FUNCTION_BLOCK CylinderSA (* Composite Function Block Type *)
  (* Standard: 61499-2 *)
  (* Version 0.0, 5/26/2016, Andrei, nxtControl GmbH, template *)
  PACKAGE Main;
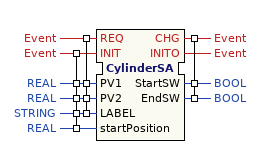
  EVENT_INPUT
    REQ WITH PV1, PV2, LABEL; (* Normal Execution Request *)
    INIT WITH PV1, PV2, LABEL, startPosition; (* Initialization Request *)
  END_EVENT
  EVENT_OUTPUT
    CHG WITH StartSW, EndSW;
    INITO; (* Initialization Confirm *)
  END_EVENT
  VAR_INPUT
    PV1 : REAL; (* Input event qualifier *)
    PV2 : REAL;
    LABEL : STRING;
    startPosition : REAL;
  END_VAR
  VAR_OUTPUT
    StartSW : BOOL; (* Output event qualifier *)
    EndSW : BOOL;
  END_VAR
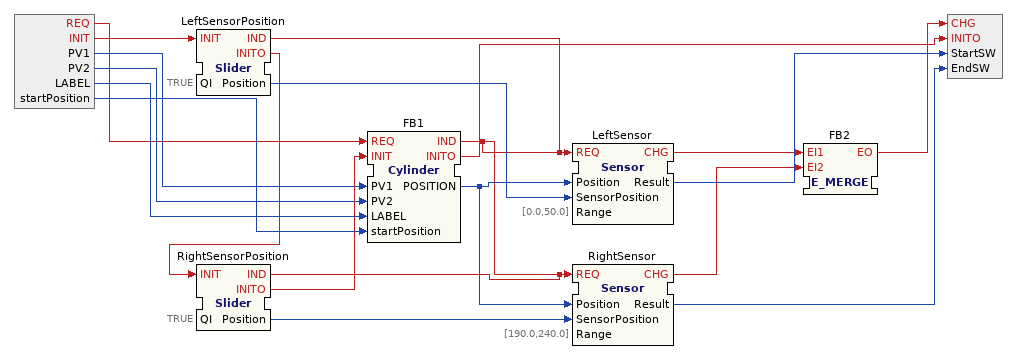
  FBS
    FB2 : E_MERGE;
    FB1 : Cylinder;
    LeftSensorPosition : Slider(QI := TRUE);
    RightSensorPosition : Slider(QI := TRUE);
    LeftSensor : Sensor(Range := [0.0,50.0]);
    RightSensor : Sensor(Range := [190.0,240.0]);
  END_FBS
  EVENT_CONNECTIONS
    REQ TO FB1.REQ;
    FB1.IND TO LeftSensor.REQ;
    FB1.IND TO RightSensor.REQ;
    LeftSensor.CHG TO FB2.EI1;
    RightSensor.CHG TO FB2.EI2;
    FB2.EO TO CHG;
    LeftSensorPosition.IND TO LeftSensor.REQ;
    RightSensorPosition.IND TO RightSensor.REQ;
    INIT TO LeftSensorPosition.INIT;
    LeftSensorPosition.INITO TO RightSensorPosition.INIT;
    RightSensorPosition.INITO TO FB1.INIT;
    FB1.INITO TO INITO;
  END_CONNECTIONS
  DATA_CONNECTIONS
    PV1 TO FB1.PV1;
    PV2 TO FB1.PV2;
    LABEL TO FB1.LABEL;
    FB1.POSITION TO LeftSensor.Position;
    FB1.POSITION TO RightSensor.Position;
    LeftSensor.Result TO StartSW;
    RightSensor.Result TO EndSW;
    LeftSensorPosition.Position TO LeftSensor.SensorPosition;
    RightSensorPosition.Position TO RightSensor.SensorPosition;
    startPosition TO FB1.startPosition;
  END_CONNECTIONS
END_FUNCTION_BLOCK
